// TIA Portal V18 export
FUNCTION "fcFonctionMathSTL" : Void   // FC3, STL
{ S7_Optimized_Access := 'TRUE' }
   VAR_INPUT
      iInputValeur1 : UDInt;
      iInputValeur2 : UDInt;
   END_VAR
   VAR_OUTPUT
      oResultValeur : UDInt;
   END_VAR
BEGIN

NETWORK
TITLE = 
      L     #iInputValeur1;
      L     #iInputValeur2;
      +D;
      T     #oResultValeur;
// Commentaire modif







END_FUNCTION
